(*
Nazwa:			E_CapFeederState
Opis:			Stany sortera nasadek
Wersja:			v0.1
Data:			2018-10-10
Autor:			DP
Urzadzenia:		
Konfiguracja:	
Info:
*)


TYPE E_CapFeederState :
(
	eDisabled:=0,  		//Wyłączona
	eError:=1,			//Błąd
	eManualMovement:=2, //Tryb serwisowy
	eHoming:=3,			//Bazowanie
	eHomingDone:=4, 	//Koniec bazowania
	eReady:=5,			//Gotowość
	eSleeveLowLevel:=6, //Praca, Niski poziom
	eSorting:=7,		//Praca
	eSleeveFull:=8,		//Zapełniona
	ePreparingToDisable:=10 (*NOWY*) //Przygotowanie do wyłączenia
):=eDisabled;
END_TYPE

(* stored: Version 1.1.0.1, ProductVersion 3.1.4026.13, FileIdentifier 876055ed545cfecc26c9384327c9d6349ce49fa5, FileSignature 8b378bc112f3053b61ebfa6ab4b69cdbe633b23b866115b28029c679ec46f7106c6d32ac59d5dd3a50c4dfb661762b9ff1335f849eafa20fcd623d87ca9e5926ba0f75ae0230eac0d56a97937be09bfb896195c4952036c57051813ee22b24bfec796ae484b4be037af8cae39910119111ccde7f9e64f4001b58f92a60551c4d4a8d4b82cd356f37931f9dabf85c701f5efa3bc7f2c6e742c40eeacca80100c299cc6dd8905b1baaece08e03079aa33480d16b81c3c0c9c6cd9b3545774ae4cb38b3be68358fa5d74b6f4e6453ed6bebfad83285101d98b700a73c8b47765c57b400d00381688626adae243aeea6907addfcc1cc00038d6a9e70935d049668f7
   DUT E_CapFeederState: Id {f0a35ac6-ab91-47de-987f-b8addf7038fd} *)
